(* IEC 61131-3 sources: generating_plc_code_with_llms/Code#2/Bard/first run, 21 files *)

(* ---- 14.st ---- *)
// 7.1s
// 2
FUNCTION FC1001 : BOOL
VAR_INPUT
    MEW : REAL;
    SP : REAL;
    HYS : REAL;
END_VAR
VAR_IN_OUT
    OUT : BOOL;
END_VAR
VAR
    P_HYS : REAL;
END_VAR

START

    P_HYS := HYS * SP;

    IF MEW > SP + P_HYS THEN
        OUT := TRUE;
    ELSIF MEW < SP - P_HYS THEN
        OUT := FALSE;
    END_IF;

    RETURN OUT;
END_FUNCTION

(* ---- 15.st ---- *)
// 8.03s
// 2
FUNCTION FC1002 : BOOL
VAR_INPUT
    E_A : BOOL;
    SENSOR : BOOL;
    ZEITW : TIME;
END_VAR
VAR_IN_OUT
    ZEIT : TON;
    P_HU : BOOL;
    P_AL : BOOL;
END_VAR

START

    IF (E_A = TRUE) AND (SENSOR = TRUE) THEN
        ZEIT := 0;
    ELSIF ZEIT > 3 THEN
        P_HU := FALSE;
        P_AL := TRUE;
    ELSIF ZEIT = 3 THEN
        P_HU := FALSE;
    ELSE
        IF ZEIT > 0 THEN
            ZEIT := ZEIT + 1;
        ELSE
            P_HU := TRUE;
        END_IF;
    END_IF;

    RETURN P_AL;
END_FUNCTION

(* ---- 18.st ---- *)
// 7.39s
// 4
FUNCTION FC1003 : VOID
VAR_INPUT
  IN_R: REAL;
  IN_MAX, IN_MIN: REAL;
  OUT_MAX, OUT_MIN: REAL;
END_VAR
VAR_OUTPUT
  OUT_R: REAL;
  FEH: BOOL;
END_VAR
VAR_TEMP
  DIFF1, DIFF2: REAL;
END_VAR

START
    DIFF1 := IN_MAX - IN_MIN;
    DIFF2 := OUT_MAX - OUT_MIN;

    IF IN_R < IN_MIN THEN
        Feh := TRUE;
        OUT_R := OUT_MIN;
    ELSIF IN_R > IN_MAX THEN
        Feh := TRUE;
        OUT_R := OUT_MAX;
    ELSE
        Feh := FALSE;
        OUT_R := (IN_R - IN_MIN) * DIFF2 / DIFF1 + OUT_MIN;
    END_IF;
END_START

(* ---- 19.st ---- *)
// 8.59s
// 3
FUNCTION_BLOCK FB1005
VAR_INPUT
  START: BOOL;
  DIKKE: REAL;
  V_MAX: REAL;
  V_MIN: REAL;
END_VAR
VAR_OUTPUT
  D_MAX: REAL;
  D_MIN: REAL;
  P1: BOOL;
END_VAR
VAR
  FO: BOOL;
END_VAR

START

    IF START = TRUE THEN
        FO := TRUE;
        D_MAX := DIKKE;
        D_MIN := DIKKE;
    ELSE
        FO := FALSE;
    END_IF;

    IF FO = TRUE THEN
        IF DIKKE > D_MAX THEN
            D_MAX := DIKKE;
        ELSIF DIKKE < D_MIN THEN
            D_MIN := DIKKE;
        END_IF;

        IF D_MAX > V_MAX THEN
            P1 := TRUE;
        ELSIF D_MIN < V_MIN THEN
            P1 := TRUE;
        ELSE
            P1 := FALSE;
        END_IF;
    END_IF;
END_START

(* ---- 20.st ---- *)
// 9.15s
// 2
FUNCTION_BLOCK INTERLOCK
VAR_INPUT
  I1 : BOOL;
  I2 : BOOL;
  TL : TIME;
END_VAR
VAR_OUTPUT
  Q1 : BOOL;
  Q2 : BOOL;
END_VAR
VAR
  T1 : TOF;
  T2 : TOF;
END_VAR

START

  IF I1 = TRUE AND Q2 = FALSE THEN
    T1 := TL;
    Q1 := TRUE;
  END_IF;

  IF I2 = TRUE AND Q1 = FALSE THEN
    T2 := TL;
    Q2 := TRUE;
  END_IF;

  IF T1 > 0 THEN
    Q1 := FALSE;
  END_IF;

  IF T2 > 0 THEN
    Q2 := FALSE;
  END_IF;
END_START

(* ---- 21.st ---- *)
// 26.65s
// 13.56s
// 2
FUNCTION_BLOCK BURNER
VAR_INPUT
  IN : BOOL;
  STAGE2 : BOOL;
  OVER_TEMP : BOOL;
  OIL_TEMP : BOOL := TRUE;
  FLAME : BOOL;
  RST : BOOL;
  RST_TIMER : BOOL;
  PRE_HEAT_TIME : TIME := t#5s;
  PRE_VENT_TIME : TIME := t#15s;
  PRE_IGNITE_TIME : TIME := t#15s;
  POST_IGNITE_TIME : TIME := t#25s;
  STAGE2_DELAY : TIME := t#10s;
  SAFETY_TIME : TIME := t#5s;
  LOCKOUT_TIME : TIME := t#10s;
  MULTIPLE_IGNITION : BOOL := TRUE;
  KW1 : REAL;
  KW2 : REAL;
END_VAR
VAR_OUTPUT
  MOTOR : BOOL;
  COIL1 : BOOL;
  COIL2 : BOOL;
  PRE_HEAT : BOOL;
  IGNITE : BOOL;
  FAIL : BOOL;
  KWH : REAL;
  STATUS : BYTE;
END_VAR
VAR_IN_OUT
  RUNTIME1 : UDINT;
  RUNTIME2 : UDINT;
  CYCLES : UDINT;
END_VAR
VAR
  state : INT;
  last : TIME;
  tx : TIME;
  last_change : TIME;
  timer1 : TON;
  timer2 : TON;
  oil_temp_last : BOOL;
  cycles2 : UDINT;
END_VAR

START

  IF RST AND RST_TIMER = FALSE THEN
    state := 0;
    timer1 := t#0s;
    timer2 := t#0s;
    cycles2 := 0;
  END_IF;

  IF OVER_TEMP THEN
    state := 0;
    FAIL := TRUE;
    STATUS := 9;
  ELSE
    IF IN AND OVER_TEMP = FALSE THEN
      IF state = 0 THEN
        // Standby
        STATUS := 110;
        IF RST_TIMER = FALSE THEN
          state := 1;
          timer1 := PRE_HEAT_TIME;
          last := TIME_OF_DAY;
        END_IF;
      ELSIF state = 1 THEN
        // Pre-heating
        PRE_HEAT := TRUE;
        IF timer1 > 0 THEN
          FAIL := NOT OIL_TEMP AND TIME_OF_DAY - last >= PRE_HEAT_TIME;
          IF FAIL THEN
            STATUS := 1;
            state := 0;
          END_IF;
        ELSE
          state := 2;
          timer1 := PRE_VENT_TIME;
          last := TIME_OF_DAY;
          MOTOR := TRUE;
        END_IF;
      ELSIF state = 2 THEN
        // Pre-ventilation
        IF timer1 > 0 THEN
          FAIL := FLAME AND TIME_OF_DAY - last >= PRE_VENT_TIME;
          IF FAIL THEN
            STATUS := 3;
            state := 0;
          END_IF;
        ELSE
          state := 3;
          timer1 := PRE_IGNITE_TIME;
          last := TIME_OF_DAY;
          IGNITE := TRUE;
        END_IF;
      ELSIF state = 3 THEN
        // Pre-ignition
        IF timer1 > 0 THEN
          FAIL := NOT FLAME AND TIME_OF_DAY - last >= PRE_IGNITE_TIME;
          IF FAIL THEN
            STATUS := 4;
            state := 0;
          END_IF;
        ELSE
          state := 4;
          timer1 := SAFETY_TIME;
          last := TIME_OF_DAY;
          COIL1 := TRUE;
        END_IF;
      ELSIF state = 4 THEN
        // Ignition
        IF timer1 > 0 THEN
          FAIL := NOT FLAME AND TIME_OF_DAY - last >= SAFETY_TIME;
          IF FAIL THEN
            STATUS := 4;
            state := 0;
          END_IF;
        ELSE
          state := 5;
          timer1 := POST_IGNITE_TIME;
          last := TIME_OF_DAY;
          tx := TIME_OF_DAY;
          KWH := 0;
        END_IF;
      ELSIF state =  5 THEN
        // Post-ignition
        IF timer1 > 0 THEN
          KWH := KW1 * (TIME_OF_DAY - tx);
        ELSE
          state := 6;
          RUNTIME1 := RUNTIME1 + TIME_OF_DAY - tx;
          IF STAGE2 AND CYCLES2 < 2 THEN
            cycles2 := cycles2 + 1;
            timer2 := STAGE2_DELAY;
            state := 7;
          ELSE
            COIL2 := TRUE;
          END_IF;
        END_IF;
      ELSIF state = 6 THEN
        // Stage 1
        RUNTIME1 := RUNTIME1 + TIME_OF_DAY - tx;
        KWH := KWH + KW1 * (TIME_OF_DAY - tx);
        IF NOT FLAME OR OVER_TEMP THEN
          state := 0;
          FAIL := TRUE;
          IF NOT FLAME THEN
            STATUS := 5;
          END_IF;
        ELSIF STAGE2 THEN
          cycles2 := cycles2 + 1;
          timer2 := STAGE2_DELAY;
          state := 7;
        END_IF;
      ELSIF state = 7 THEN
        // Stage 2 delay
        IF timer2 > 0 THEN
          // Do nothing, wait for timer
        ELSE
          state := 8;
          COIL2 := TRUE;
        END_IF;
      ELSIF state = 8 THEN
        // Stage 2
        RUNTIME2 := RUNTIME2 + TIME_OF_DAY - tx;
        KWH := KWH + KW2 * (TIME_OF_DAY - tx);
        IF NOT FLAME OR OVER_TEMP THEN
          state := 0;
          FAIL := TRUE;
          IF NOT FLAME THEN
            STATUS := 5;
          END_IF;
        END_IF;
      END_IF;

IF RST AND RST_TIMER = FALSE THEN
  RST_TIMER := TRUE;
  timer1 := LOCKOUT_TIME;
END_IF;

IF RST_TIMER > 0 THEN
  STATUS := 0;
END_IF;

END_START

(* ---- 1.st ---- *)
// 5.13s
// 4
VAR
    xAllOn : BOOL;
    xAllOff : BOOL;

    xAlarm1 : BOOL;
    xAlarm2 : BOOL;
END_VAR

START

    IF xAllOn THEN
        xAlarm1 := TRUE;
        xAlarm2 := TRUE;
        xAllOn := FALSE;
    END_IF;

    IF xAllOff THEN
        xAlarm1 := FALSE;
        xAlarm2 := FALSE;
        xAllOff := FALSE;
    END_IF;

END_START

(* ---- 10.st ---- *)
// 5.63s
// 4
VAR
    Y : REAL;
END_VAR

START

    Y := 1.0 / (1.0 + exp(-X));
END_START

(* ---- 11.st ---- *)
// 5.49s
// 4
VAR
    Y : REAL;
END_VAR

START

    IF x < 0 THEN
        Y := -1.0;
    ELSIF x = 0 THEN
        Y := 0.0;
    ELSE
        Y := 1.0;
    END_IF;
END_START

(* ---- 12.st ---- *)
// 6.31s
// 3
VAR
    Y : REAL;
END_VAR

START

    Y := exp(X) + exp(-X);
END_START

(* ---- 13.st ---- *)
// 8.17s
// 2
VAR CONSTANT
    MAXNUMBERS : UINT := 99;
END_VAR

VAR
    aNumbers : ARRAY[0..MAXNUMBERS] OF INT;
    nSearchNumber : INT;
    nCnt : INT;
END_VAR

START

    nSearchNumber := 50;

    REPEAT
        nCnt := nCnt + 1;

        IF aNumbers[nCnt] = nSearchNumber THEN
            EXIT;
        ELSIF aNumbers[nCnt] = 10 THEN
            EXIT;
        END_IF;
    END_REPEAT;

    IF nCnt = MAXNUMBERS THEN
        nCnt := -1;
    END_IF;
END_START

(* ---- 16.st ---- *)
// 8.59s
// 2
VAR
  North_green : BOOL;
  North_yellow : BOOL;
  North_red : BOOL;
  East_green : BOOL;
  East_yellow : BOOL;
  East_red : BOOL;
  T1 : TON;
END_VAR

START

  T1 := 0;

  North_green := TRUE;
  North_yellow := FALSE;
  North_red := FALSE;
  East_green := FALSE;
  East_yellow := FALSE;
  East_red := TRUE;

  WHILE T1 < 5000 DO

    IF T1 >= 4500 THEN
      North_green := FALSE;
      North_yellow := TRUE;
    END_IF;

    IF T1 >= 5500 THEN
      North_yellow := FALSE;
      North_red := TRUE;
      East_green := TRUE;
      East_red := FALSE;
    END_IF;

    IF T1 >= 9500 THEN
      East_green := FALSE;
      East_yellow := TRUE;
    END_IF;

    IF T1 >= 10000 THEN
      East_yellow := FALSE;
      East_red := TRUE;
    END_IF;

    END_WHILE;

END_START

(* ---- 17.st ---- *)
// 7.17s
// 2
VAR
  aiOutside : INT;
  aiHumidity: INT;
  sShowText : STRING[80];
END_VAR

START

    aiOutside := ReadAnalogInput();
    aiHumidity := ReadAnalogInput();

    IF (aiOutside < 18) THEN
        sShowText := "Cold";
    ELSIF (aiOutside <= 25) AND (aiHumidity >= 40) AND (aiHumidity <= 75) THEN
        sShowText := "Opt";
    ELSIF (aiOutside <= 25) AND (aiHumidity < 40) OR (aiHumidity > 75) THEN
        sShowText := "Temp. OK";
    ELSE
        sShowText := "Hot";
    END_IF;

    DisplayText(sShowText);
END_START

(* ---- 2.st ---- *)
// 4.87s
// 3
VAR_INPUT
    N : INT;
    K : INT;
    i : INT;
END_VAR

VAR
    binomialCoefficient : INT := 1;
END_VAR

START

    FOR i := 0 TO K DO
        binomialCoefficient := binomialCoefficient * (N - i) / i;
    END_FOR;

END_START

(* ---- 3.st ---- *)
// 5.01s
// 2
VAR_INPUT
    X : INT;
END_VAR
VAR
    t1 : DINT;
    t2 : DINT;
    y_tmp : INT;
END_VAR

START

    IF X = 0 THEN
        Y := 0;
    ELSIF X = 1 THEN
        Y := 1;
    ELSE
        Y := 0;
        x_tmp := 1;
        t1 := 1;

        FOR i := 2 TO X DO
            Y := Y + x_tmp;
            t2 := t1;
            t1 := Y;
            x_tmp := t2;
        END_FOR;
    END_IF;

END_START

(* ---- 4.st ---- *)
// 6.45s
// 2
VAR
    aiLevel : INT;
    PercentLevel : UINT;
    doLow : BOOL;
    doOk : BOOL;
    doHigh : BOOL;
    doAlarm : BOOL;
END_VAR

START

    READ_ANALOG aiLevel;

    IF aiLevel < 0 THEN
        PercentLevel := 0;
    ELSE
        IF aiLevel > 32767 THEN
            PercentLevel := 100;
        ELSE
            PercentLevel := INT((aiLevel) * 100 / 32767);
        END_IF;
    END_IF;

    CASE PercentLevel
        WHEN 0..25 THEN
            doLow := TRUE;
            doOk := FALSE;
            doHigh := FALSE;
            doAlarm := FALSE;
        WHEN 26..75 THEN
            doLow := FALSE;
            doOk := TRUE;
            doHigh := FALSE;
            doAlarm := FALSE;
        WHEN 76..100 THEN
            doLow := FALSE;
            doOk := FALSE;
            doHigh := TRUE;
            doAlarm := FALSE;
        ELSE
            doLow := FALSE;
            doOk := FALSE;
            doHigh := FALSE;
            doAlarm := TRUE;
    END_CASE;

END_START

(* ---- 5.st ---- *)
// 7.62s
// 2
VAR
    Start_Loop : BOOL := FALSE;
    one_hour : TIME := T#1h;
    One_Hour_Timer : TON;
    Gate_Open : BOOL := FALSE;
    Close_Gate_Inst : BOOL := FALSE;
    Sensed_Car : BOOL := FALSE;
    Sensed_Car_Inst : BOOL := FALSE;
    Sensed_App : BOOL := FALSE;
    Mobile_Inst : BOOL := FALSE;
    Auth : STRING;
    my_defined_str : STRING := 'abcd';
END_VAR

START

    IF Start_Loop = TRUE THEN
        Close_Gate_Inst := TRUE;
    END_IF;

    IF Sensed_Car = TRUE THEN
        IF Auth = my_defined_str THEN
            Gate_Open := TRUE;
            Close_Gate_Inst := FALSE;
        END_IF;
    END_IF;

    IF Mobile_Inst = TRUE THEN
        IF Auth = my_defined_str THEN
            Gate_Open := TRUE;
            Close_Gate_Inst := FALSE;
        END_IF;
    END_IF;

    IF NOT Gate_Open AND Close_Gate_Inst THEN
        Close_Gate_Inst := FALSE;
        IF One_Hour_Timer.Q THEN
            Gate_Open := FALSE;
        ELSE
            One_Hour_Timer.Start(one_hour);
        END_IF;
    END_IF;

    One_Hour_Timer.RUN := Start_Loop;

END_START

(* ---- 6.st ---- *)
// 9.91s
// 2
VAR CONSTANT
    WAIT : UINT := 0;
    TOP_POSITION : UINT := 1;
    BOTTOM_POSITION : UINT := 2;
    GETBOX : UINT := 3;
    UNLOAD_POSITION : UINT := 4;
    UNLOAD_BOX : UINT := 5;
END_VAR

VAR
    (*-- digital outputs*)
    doConvTop: BOOL := FALSE;
    doConvBottom: BOOL := FALSE;
    doConvLift: BOOL := FALSE;
    doLiftTop: BOOL := FALSE;
    doLiftBottom: BOOL := FALSE;
    doLiftUnload: BOOL := FALSE;
    (*-- digital inputs*)
    diConvTop: BOOL := FALSE;
    diConvBottom: BOOL := FALSE;
    diLiftTop: BOOL := FALSE;
    diLiftBottom: BOOL := FALSE;
    diLiftUnload: BOOL := FALSE;
    diBoxLift: BOOL := FALSE;
    (*-- status variables*)
    selectLift: UINT := 0;
    ConvTopOn: BOOL := FALSE;
    ConvBottomOn: BOOL := FALSE;
END_VAR

START

    IF diConvTop THEN
        ConvTopOn := TRUE;
        doConvTop := FALSE;
        selectLift := TOP_POSITION;
    END_IF;

    IF diConvBottom THEN
        ConvBottomOn := TRUE;
        doConvBottom := FALSE;
        selectLift := BOTTOM_POSITION;
    END_IF;

    CASE selectLift
        WHEN TOP_POSITION OR BOTTOM_POSITION THEN
            IF diLiftTop AND ConvTopOn THEN
                doLiftTop := TRUE;
                selectLift := GETBOX;
            ELSIF diLiftBottom AND ConvBottomOn THEN
                doLiftBottom := TRUE;
                selectLift := GETBOX;
            END_IF;
        WHEN GETBOX THEN
            IF diBoxLift THEN
                doConvLift := TRUE;
            END_IF;
        WHEN UNLOAD_POSITION THEN
            IF diLiftUnload THEN
                doLiftUnload := TRUE;
                selectLift := UNLOAD_BOX;
            END_IF;
        WHEN UNLOAD_BOX THEN
            IF diConvTop OR diConvBottom THEN
                selectLift := WAIT;
            END_IF;
    END_CASE;

END_START

(* ---- 7.st ---- *)
// 7.63s
// 2
VAR CONSTANT
    MAX_INDEX: USINT := 4;
END_VAR
VAR
    aWeights: ARRAY[0..MAX_INDEX] OF INT;
    iCnt: USINT;
    sumWeight: DINT := 0;
    avgWeight: INT;
END_VAR

START

    FOR iCnt := 0 TO MAX_INDEX DO
        READ_ANALOG aWeights[iCnt];
        sumWeight := sumWeight + aWeights[iCnt];
    END_FOR;

    avgWeight := sumWeight / MAX_INDEX;
    WRITE_ANALOG avgWeight;

END_START

(* ---- 8.st ---- *)
// 9.07s
// 2
VAR_INPUT
    X : REAL;
END_VAR
VAR
    w : REAL;
    i : INT;
    we : REAL;
    w1e : REAL;
    ewx : REAL;
    last : DWORD;
END_VAR

START

    ewx := 1;
    we := X;
    last := 0;

    i := 1;

    WHILE ((abs(we - ewx) > 0.0001) AND (i < 100)) DO
        we := (we + ewx) / 2;

        w1e := ewx * exp(w);

        ewx := (w * we) - X;

        IF (last = 1) AND (we < 0) THEN
            ewx := 0;
        END_IF;

        last := abs(we) > abs(ewx);

        i := i + 1;
    END_WHILE;

    w := we;
END_START

(* ---- 9.st ---- *)
// 6.98s
// 2
VAR
    YEAR : INT;
END_VAR

START

    IF (YEAR % 4 = 0) AND (YEAR % 100 <> 0) OR (YEAR % 400 = 0) THEN
        LeapYear := TRUE;
    ELSE
        LeapYear := FALSE;
    END_IF;
END_START
